Omron CX-Programmer project NewProject (CX-Programmer 9.73)

# PLC NewPLC1: CP1E N20

## Global symbols (name address type ; comment)
0.01 BOOL  ; pb start
0.02 BOOL  ; rs1
0.03 BOOL  ; pb stop
0.04 BOOL  ; rs2
100.00 BOOL  ; cylinder
200.00 BOOL  ; relay

## Program NewProgram1 (cyclic task 0)

### Section Section1

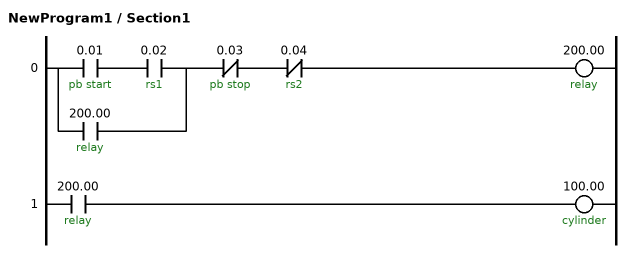
; rung 0
LD 0.01  ; pb start
AND 0.02  ; rs1
OR 200.00  ; relay
ANDNOT 0.03  ; pb stop
ANDNOT 0.04  ; rs2
OUT 200.00  ; relay
; rung 1
LD 200.00  ; relay
OUT 100.00  ; cylinder

### Section END
; rung 0
END(001)